FUNCTION_BLOCK MachineCycle EXTENDS StateMachine
VAR_INPUT
END_VAR
VAR_OUTPUT
END_VAR
VAR
END_VAR

SUPER^();
Start();

METHOD PROTECTED Busy : BOOL
VAR_INPUT
END_VAR
VAR_INST
	eAdsConnectorBusy : E_AdsConnectorBusy;
END_VAR
END_METHOD

METHOD PROTECTED  Error : BOOL
VAR_INPUT
END_VAR
END_METHOD

METHOD PROTECTED  Idle : BOOL
VAR_INPUT
END_VAR
END_METHOD

METHOD PROTECTED  Init : BOOL
VAR_INPUT
END_VAR
END_METHOD

METHOD PROTECTED  Prepare : BOOL
VAR_INPUT
END_VAR
END_METHOD

METHOD PROTECTED  Ready : BOOL
VAR_INPUT
END_VAR
(*
Check conditions to fire Execute() here and put the StateMachine in Busy mode
*)
END_METHOD

METHOD PROTECTED  Waiting : BOOL
VAR_INPUT
END_VAR
END_METHOD

END_FUNCTION_BLOCK

(* stored: Version 1.1.0.1, ProductVersion 3.1.4024.0
   POU MachineCycle: Id {fdc3671d-6149-42f8-9b1d-397b8dace8e6}, SpecialFunc None
   Method Busy: Id {5d591906-f587-4523-9091-f95c379d4cb3}
   Method Error: Id {7b29483d-0108-41c8-b9cf-998033a135d9}
   Method Idle: Id {cd2e702c-923b-4852-ab0b-3a97f38d2fa9}
   Method Init: Id {ccd6d14a-344c-4a25-bfc3-ce5e939c71cc}
   Method Prepare: Id {32a12e8b-2e91-409a-834d-b1ce78bae0e2}
   Method Ready: Id {23737be8-0a59-4a9a-8e15-4787ed54319c}
   Method Waiting: Id {7b8620e8-4807-4be1-bccc-712aaca2aa48} *)
